{attribute 'qualified_only'}
VAR_GLOBAL
	
	MC_MoveAbsolute: MC_MoveAbsolute;
	MC_MoveAbsolute_output: ST_McOutputs;
END_VAR

(* stored: Version 1.1.0.1, ProductVersion 3.1.4024.9
   GVL GVL: Id {7781904d-981b-482e-8d45-f20f49e1ec75} *)
